// TIA Portal V17 export
// export: Created 2022-07-28T18:02:45.2636855Z, ExportSetting None, DisplayName Totally Integrated Automation Portal, DisplayVersion V17, DisplayName TIA Portal Openness, DisplayVersion V17, DisplayName TIA Portal Teamcenter Gateway, DisplayVersion V17, DisplayName TIA Portal Version Control Interface, DisplayVersion V17, DisplayName TIA Portal Test Suite Advanced, DisplayVersion V17, DisplayName SINAMICS Startdrive Advanced, DisplayVersion V17, DisplayName SINAMICS DCC, DisplayVersion V17, DisplayName SINAMICS Startdrive G130, G150, S120, S150, SINAMICS MV, S210, DisplayVersion V17, DisplayName SINAMICS Startdrive G110M, G120, G120C, G120D, G120P, G115D, DisplayVersion V17, DisplayName STEP 7 Professional, DisplayVersion V17, DisplayName SIMATIC Energy Suite, DisplayVersion V17, DisplayName STEP 7 CFC, DisplayVersion V17, DisplayName STEP 7 Safety, DisplayVersion V17, DisplayName WinCC Advanced / Unified PC, DisplayVersion V17, DisplayName SIMATIC Visualization Architect, DisplayVersion V17
FUNCTION "Lib_FC_General_CountMotoHours" : Void   // FC10, SCL
{ S7_Optimized_Access := 'TRUE' }
// stored: SetENOAutomatically false
   VAR_INPUT
      II_Obj_ID : Int;   // Tech ID of object
      I_One_1s : Bool;   // 1 = One cycle per one seccond pulse
      I_Run : Bool;   // 1 = Motor running
      I_PosPulseSimMode : Bool;   // 1 = Once when enter into simulation mode
      I_NegPulseSimMode : Bool;   // 1 = Once when exit from simulation mode
   END_VAR
   VAR_OUTPUT
      Q_MaintenanceElectroServ : Bool;   // x2 - 1 = [3-level ] - Maintenance - Обслуговування - Спрацювали таймери/лічильники обслуговування
      Q_MaintenanceMechanoServ : Bool;   // x2 - 1 = [3-level ] - Maintenance - Обслуговування - Спрацювали таймери/лічильники обслуговування
   END_VAR
   VAR_IN_OUT
      IQUD_BacUpElectro : "_MotoHours_One";   // Backup buffer for simulation mode for motohours
      IQUD_BacUpMechanic : "_MotoHours_One";   // Backup buffer for simulation mode for motohours
   END_VAR
   VAR_TEMP
      ti_Count : Int;   // Counter for loop
      tud_MotoHours_Electro : "_MotoHours_One";
      tud_MotoHours_Mech : "_MotoHours_One";
      t_MaintenanceElectroServ : Bool;   // x2 - 1 = [3-level ] - Maintenance - Обслуговування - Спрацювали таймери/лічильники обслуговування
      t_MaintenanceMechanoServ : Bool;   // x2 - 1 = [3-level ] - Maintenance - Обслуговування - Спрацювали таймери/лічильники обслуговування
      t_MaxObjects : UInt;   // Max number of objects in plant
   END_VAR
BEGIN
   //Read general info data
   #t_MaxObjects := "D_General_ProgramDATA".ui_MaxObjects;
   #tud_MotoHours_Electro := "D_General_MotoHours_Electro".Arr[#t_MaxObjects];
   #tud_MotoHours_Mech := "D_General_MotoHours_Mech".Arr[#t_MaxObjects];

   CASE #II_Obj_ID OF
       0..999:  // ID of element in range
           #tud_MotoHours_Electro := "D_General_MotoHours_Electro".Arr[#II_Obj_ID];
           #tud_MotoHours_Mech := "D_General_MotoHours_Mech".Arr[#II_Obj_ID];
       ELSE
           ;
   END_CASE;
   //---------------------------------------------------------------
   //---------------------------------------------------------------
   REGION Work with backup for simulation mode
       IF #I_PosPulseSimMode
       THEN
           #IQUD_BacUpElectro := #tud_MotoHours_Electro;
           #IQUD_BacUpMechanic := #tud_MotoHours_Mech;
       END_IF;

       IF #I_NegPulseSimMode
       THEN
           #tud_MotoHours_Electro := #IQUD_BacUpElectro;
           #tud_MotoHours_Mech := #IQUD_BacUpMechanic;
           #IQUD_BacUpElectro := "D_General_MotoHours_Electro".Arr[#t_MaxObjects];
           #IQUD_BacUpMechanic := "D_General_MotoHours_Mech".Arr[#t_MaxObjects];
       END_IF;
   END_REGION
   //---------------------------------------------------------------
   //---------------------------------------------------------------
   REGION Count motohours
       //Reinit bits
       #t_MaintenanceElectroServ := false;
       #t_MaintenanceMechanoServ := false;

       //Loop through all SP
       FOR #ti_Count := 1 TO 7 DO
           REGION Count actual motohourses
               IF #I_One_1s
                   AND #I_Run
               THEN
                   //For electroservice
                   IF #tud_MotoHours_Electro.Arr[#ti_Count].di_SetMotoHours > 0
                   THEN
                       #tud_MotoHours_Electro.Arr[#ti_Count].di_ActMotoHours += 1;
                   END_IF;

                   //For mechanoservice
                   IF #tud_MotoHours_Mech.Arr[#ti_Count].di_SetMotoHours > 0
                   THEN
                       #tud_MotoHours_Mech.Arr[#ti_Count].di_ActMotoHours += 1;
                   END_IF;
               END_IF;
           END_REGION
           //---------------------------------------------------------------
           //---------------------------------------------------------------
           REGION Reset counters
               //For electroservice
               IF (#tud_MotoHours_Electro.i_CMD = (50 + #ti_Count - 1))
                   OR (#tud_MotoHours_Electro.Arr[#ti_Count].di_SetMotoHours <= 0)
               THEN
                   #tud_MotoHours_Electro.Arr[#ti_Count].di_ActMotoHours := 0;
                   #tud_MotoHours_Electro.i_CMD := 0;
               END_IF;

               //For mechanoservice
               IF (#tud_MotoHours_Mech.i_CMD = (50 + #ti_Count - 1))
                   OR (#tud_MotoHours_Mech.Arr[#ti_Count].di_SetMotoHours <= 0)
               THEN
                   #tud_MotoHours_Mech.Arr[#ti_Count].di_ActMotoHours := 0;
                   #tud_MotoHours_Mech.i_CMD := 0;
               END_IF;

           END_REGION
           //---------------------------------------------------------------
           //---------------------------------------------------------------
           REGION Set maintenance alarm
               //For electroservice
               #tud_MotoHours_Electro.Arr[#ti_Count].di_ActLeftMotoHours := #tud_MotoHours_Electro.Arr[#ti_Count].di_SetMotoHours
               - #tud_MotoHours_Electro.Arr[#ti_Count].di_ActMotoHours;

               IF #tud_MotoHours_Electro.Arr[#ti_Count].di_ActLeftMotoHours <= 0
                   AND #tud_MotoHours_Electro.Arr[#ti_Count].di_SetMotoHours > 0
               THEN
                   #t_MaintenanceElectroServ := true;
               END_IF;

               //For mechanoservice
               #tud_MotoHours_Mech.Arr[#ti_Count].di_ActLeftMotoHours := #tud_MotoHours_Mech.Arr[#ti_Count].di_SetMotoHours
               - #tud_MotoHours_Mech.Arr[#ti_Count].di_ActMotoHours;

               IF #tud_MotoHours_Mech.Arr[#ti_Count].di_ActLeftMotoHours <= 0
                   AND #tud_MotoHours_Mech.Arr[#ti_Count].di_SetMotoHours > 0
               THEN
                   #t_MaintenanceMechanoServ := true;
               END_IF;
           END_REGION

       END_FOR;
   END_REGION
   //---------------------------------------------------------------
   //---------------------------------------------------------------
   REGION Outputs of block
       #Q_MaintenanceElectroServ := #t_MaintenanceElectroServ;
       #Q_MaintenanceMechanoServ := #t_MaintenanceMechanoServ;
   END_REGION
   //---------------------------------------------------------------
   //---------------------------------------------------------------
   //Write general info data
   CASE #II_Obj_ID OF
       0..999:  // ID of element in range
           "D_General_MotoHours_Electro".Arr[#II_Obj_ID] := #tud_MotoHours_Electro;
           "D_General_MotoHours_Mech".Arr[#II_Obj_ID] := #tud_MotoHours_Mech;
       ELSE
           ;
   END_CASE;
END_FUNCTION
